FUNCTION_BLOCK TestPOU
VAR_INPUT
	FirstIntput : BOOL;
	SecondInput : BOOL;
	_SecondInput : BOOL;
	s_SecondInput : BOOL;
END_VAR
VAR_OUTPUT
END_VAR
VAR
END_VAR

END_FUNCTION_BLOCK

(* stored: Version 1.1.0.1, ProductVersion 3.1.4024.6
   POU TestPOU: Id {e9284524-1b8f-4e59-87db-04d925e94940}, SpecialFunc None *)
